// SIMATIC STEP 7 (V5.x) project TEMA 8 EJRCICIO 4
// CPU: CPU313 C-2 DP(1)
// station: P_ADR_BUS
// station: Hardware
// station: Equipo SIMATIC 300
// program: Programa S7(1)

SYMBOL_TABLE
"F CARRERA"	DB 1	DB 1
"MANIOBRA"	DB 2	DB 2
"ENCLAVAMIENTO"	DB 3	DB 3
"S LENTO"	I 0.0	BOOL
"S RAPIDO"	I 0.1	BOOL
"B LENTO"	I 0.2	BOOL
"B RAPIDO"	I 0.3	BOOL
"D LENTO"	I 0.4	BOOL
"D RAPIDO"	I 0.5	BOOL
"I LENTO"	I 0.6	BOOL
"I RAPIDO"	I 0.7	BOOL
"FC BAJADA"	I 1.0	BOOL
"FC SUBIDA"	I 1.1	BOOL
"FC IZQUIERDA"	I 1.2	BOOL
"FC DERECHA"	I 1.3	BOOL
"Cycle Execution"	OB 1	OB 1
"M1S U1-V1-W1TSR"	Q 0.0	BOOL
"M1S U2-V2-W2TSR"	Q 0.1	BOOL
"M1SB CORTOCIRCUITADO"	Q 0.2	BOOL
"M1B U1-V1-W1RST"	Q 0.3	BOOL
"M1B U2-V2-W2RST"	Q 0.4	BOOL
"M2D U1-V1-W1RST"	Q 0.5	BOOL
"M2D U2-V2-W2RST"	Q 0.6	BOOL
"M2DI CORTOCIRCUITADO"	Q 0.7	BOOL
"M2I U1-V1-W1TSR"	Q 1.0	BOOL
"M2I U2-V2-W2 TSR"	Q 1.1	BOOL
"VAT_1"	VAT 1	
END_SYMBOL_TABLE

DATA_BLOCK "F CARRERA"	// DB 1
VERSION : 0.1
  STRUCT
   BAJADA : BOOL ;
   SUBIDA : BOOL ;
   IZQUIERDA : BOOL ;
   DERECHA : BOOL ;
  END_STRUCT ;	
BEGIN
END_DATA_BLOCK

DATA_BLOCK "MANIOBRA"	// DB 2
VERSION : 0.1
  STRUCT
   MARCA0 : BOOL ;
   MARCA1 : BOOL ;
   MARCA2 : BOOL ;
   MARCA3 : BOOL ;
   MARCA4 : BOOL ;
   MARCA5 : BOOL ;
   MARCA6 : BOOL ;
   MARCA7 : BOOL ;
  END_STRUCT ;	
BEGIN
END_DATA_BLOCK

DATA_BLOCK "ENCLAVAMIENTO"	// DB 3
VERSION : 0.1
  STRUCT
   SUBIDA : BOOL ;
   BAJADA : BOOL ;
   DERECHA : BOOL ;
   IZQUIERDA : BOOL ;
  END_STRUCT ;	
BEGIN
END_DATA_BLOCK

ORGANIZATION_BLOCK "Cycle Execution"	// OB 1
TITLE = "Main Program Sweep (Cycle)"
//PUENTE GRUA CON DOS VELOCIDADES A IMPULSOS .NO PUEDEN FUNCIONAR A LA VEZ 2 
//VELOCIDADES DEL MISMO SENTIDO Y TAMPOCO DOS DIRECCIONES DEL MISMO MOTOR
VERSION : 0.1
VAR_TEMP
  OB1_EV_CLASS : BYTE ;	//Bits 0-3 = 1 (Coming event), Bits 4-7 = 1 (Event class 1)
  OB1_SCAN_1 : BYTE ;	//1 (Cold restart scan 1 of OB 1), 3 (Scan 2-n of OB 1)
  OB1_PRIORITY : BYTE ;	//Priority of OB Execution
  OB1_OB_NUMBR : BYTE ;	//1 (Organization block 1, OB1)
  OB1_RESERVED_1 : BYTE ;	//Reserved for system
  OB1_RESERVED_2 : BYTE ;	//Reserved for system
  OB1_PREV_CYCLE : INT ;	//Cycle time of previous OB1 scan (milliseconds)
  OB1_MIN_CYCLE : INT ;	//Minimum cycle time of OB1 (milliseconds)
  OB1_MAX_CYCLE : INT ;	//Maximum cycle time of OB1 (milliseconds)
  OB1_DATE_TIME : DATE_AND_TIME ;	//Date and time OB1 started
END_VAR
BEGIN
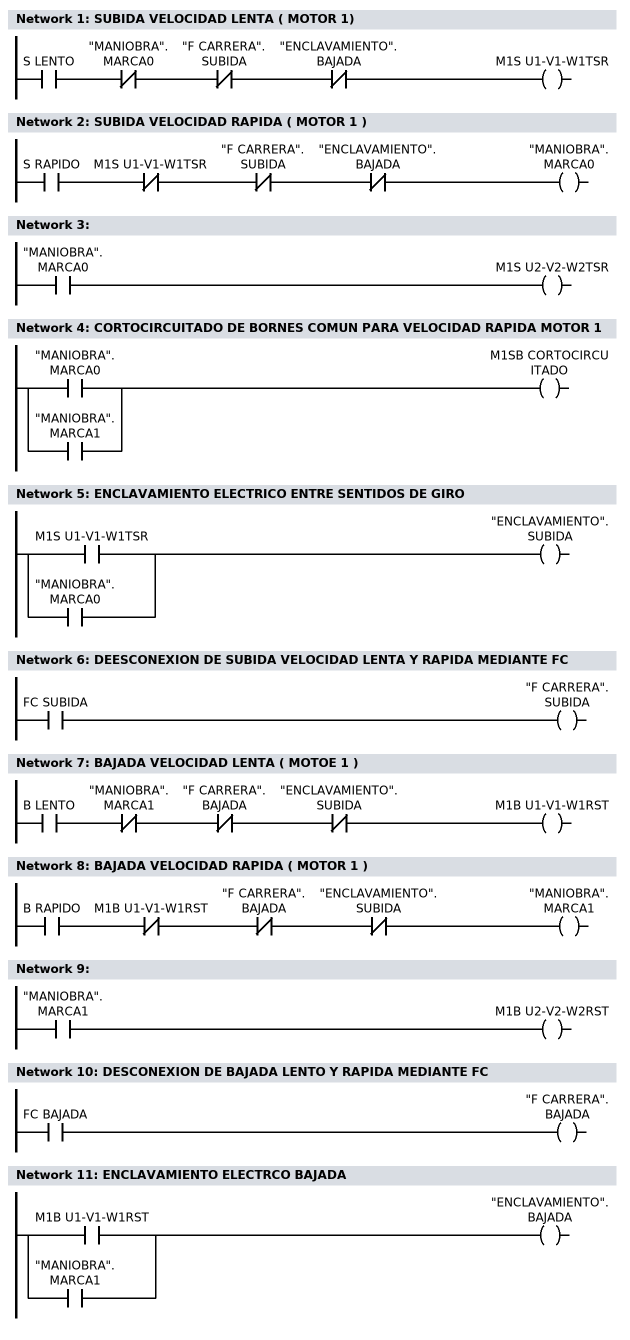
NETWORK
TITLE = SUBIDA VELOCIDAD LENTA ( MOTOR 1)
      A     "S LENTO";
      AN    "MANIOBRA".MARCA0;
      AN    "F CARRERA".SUBIDA;
      AN    "ENCLAVAMIENTO".BAJADA;
      =     "M1S U1-V1-W1TSR";
NETWORK
TITLE = SUBIDA VELOCIDAD RAPIDA ( MOTOR 1 )
      A     "S RAPIDO";
      AN    "M1S U1-V1-W1TSR";
      AN    "F CARRERA".SUBIDA;
      AN    "ENCLAVAMIENTO".BAJADA;
      =     "MANIOBRA".MARCA0;
NETWORK
TITLE =
      A     "MANIOBRA".MARCA0;
      =     "M1S U2-V2-W2TSR";
NETWORK
TITLE = CORTOCIRCUITADO DE BORNES COMUN PARA VELOCIDAD RAPIDA MOTOR 1
      O     "MANIOBRA".MARCA0;
      O     "MANIOBRA".MARCA1;
      =     "M1SB CORTOCIRCUITADO";
NETWORK
TITLE = ENCLAVAMIENTO ELECTRICO ENTRE SENTIDOS DE GIRO
//CUANDO MOTOR 1 FUNCIONE EN SENTIDO ARRIBA TANTO EN VELOCIDAD LENTA COMO RAPIDA  
//ESTA MARCA EVITARA QUE PUEDA CONECTAR LOS 2 SENTIDOS DE GIRO A LA VEZ Y POR LO 
//TANTO PRODUCIR UN ERROR FATAL PARA MOTOR 1.SE INSERTARA UN CONTACTO CERRADO 
//ANTES DE LAS BOBINAS DEL SENTIDO CONTRARIO PARA QUE SE HABRAN Y POR LO TANTO NO 
//PODRA ALIMENTAR ESAS BOBINAS MIENTRAS ESTEN ALIMENTADAS LAS OTRAS.
// 
//
      O     "M1S U1-V1-W1TSR";
      O     "MANIOBRA".MARCA0;
      =     "ENCLAVAMIENTO".SUBIDA;
NETWORK
TITLE = DEESCONEXION DE SUBIDA VELOCIDAD LENTA Y RAPIDA MEDIANTE FC
      A     "FC SUBIDA";
      =     "F CARRERA".SUBIDA;
NETWORK
TITLE = BAJADA VELOCIDAD LENTA ( MOTOE 1 )
      A     "B LENTO";
      AN    "MANIOBRA".MARCA1;
      AN    "F CARRERA".BAJADA;
      AN    "ENCLAVAMIENTO".SUBIDA;
      =     "M1B U1-V1-W1RST";
NETWORK
TITLE = BAJADA VELOCIDAD RAPIDA ( MOTOR 1 )
      A     "B RAPIDO";
      AN    "M1B U1-V1-W1RST";
      AN    "F CARRERA".BAJADA;
      AN    "ENCLAVAMIENTO".SUBIDA;
      =     "MANIOBRA".MARCA1;
NETWORK
TITLE =
      A     "MANIOBRA".MARCA1;
      =     "M1B U2-V2-W2RST";
NETWORK
TITLE = DESCONEXION DE BAJADA LENTO Y RAPIDA MEDIANTE FC
      A     "FC BAJADA";
      =     "F CARRERA".BAJADA;
NETWORK
TITLE = ENCLAVAMIENTO ELECTRCO BAJADA
      O     "M1B U1-V1-W1RST";
      O     "MANIOBRA".MARCA1;
      =     "ENCLAVAMIENTO".BAJADA;
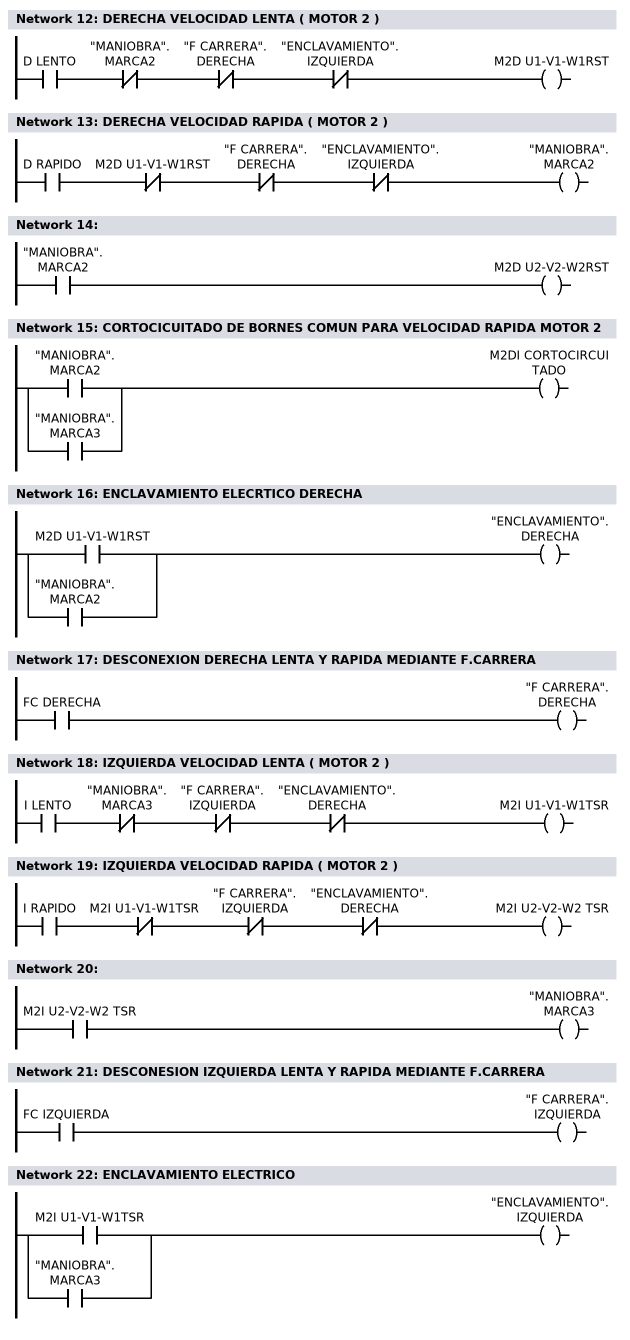
NETWORK
TITLE = DERECHA VELOCIDAD LENTA ( MOTOR 2 )
      A     "D LENTO";
      AN    "MANIOBRA".MARCA2;
      AN    "F CARRERA".DERECHA;
      AN    "ENCLAVAMIENTO".IZQUIERDA;
      =     "M2D U1-V1-W1RST";
NETWORK
TITLE = DERECHA VELOCIDAD RAPIDA ( MOTOR 2 )
      A     "D RAPIDO";
      AN    "M2D U1-V1-W1RST";
      AN    "F CARRERA".DERECHA;
      AN    "ENCLAVAMIENTO".IZQUIERDA;
      =     "MANIOBRA".MARCA2;
NETWORK
TITLE =
      A     "MANIOBRA".MARCA2;
      =     "M2D U2-V2-W2RST";
NETWORK
TITLE = CORTOCICUITADO DE BORNES COMUN PARA VELOCIDAD RAPIDA MOTOR 2
      O     "MANIOBRA".MARCA2;
      O     "MANIOBRA".MARCA3;
      =     "M2DI CORTOCIRCUITADO";
NETWORK
TITLE = ENCLAVAMIENTO ELECRTICO DERECHA
      O     "M2D U1-V1-W1RST";
      O     "MANIOBRA".MARCA2;
      =     "ENCLAVAMIENTO".DERECHA;
NETWORK
TITLE = DESCONEXION DERECHA LENTA Y RAPIDA MEDIANTE F.CARRERA
      A     "FC DERECHA";
      =     "F CARRERA".DERECHA;
NETWORK
TITLE = IZQUIERDA VELOCIDAD LENTA ( MOTOR 2 )
      A     "I LENTO";
      AN    "MANIOBRA".MARCA3;
      AN    "F CARRERA".IZQUIERDA;
      AN    "ENCLAVAMIENTO".DERECHA;
      =     "M2I U1-V1-W1TSR";
NETWORK
TITLE = IZQUIERDA VELOCIDAD RAPIDA ( MOTOR 2 )
      A     "I RAPIDO";
      AN    "M2I U1-V1-W1TSR";
      AN    "F CARRERA".IZQUIERDA;
      AN    "ENCLAVAMIENTO".DERECHA;
      =     "M2I U2-V2-W2 TSR";
NETWORK
TITLE =
      A     "M2I U2-V2-W2 TSR";
      =     "MANIOBRA".MARCA3;
NETWORK
TITLE = DESCONESION IZQUIERDA LENTA Y RAPIDA MEDIANTE F.CARRERA
      A     "FC IZQUIERDA";
      =     "F CARRERA".IZQUIERDA;
NETWORK
TITLE = ENCLAVAMIENTO ELECTRICO
      O     "M2I U1-V1-W1TSR";
      O     "MANIOBRA".MARCA3;
      =     "ENCLAVAMIENTO".IZQUIERDA;
END_ORGANIZATION_BLOCK
